FUNCTION_BLOCK FB_String_Test EXTENDS TcUnit.FB_TestSuite

WhenSubtringExistsExpectPosition();
WhenMonthToStringReturnsCorrectMonthName();

METHOD PRIVATE WhenMonthToStringReturnsCorrectMonthName
VAR
    ActualMonth : STRING(10);
    ExpectedMonth : STRING(10) := 'January';
    MTH : INT := 1;
    LANG : INT := 1; // Adjust as needed for your language table
    LX : INT := 0;
END_VAR
TEST(__POUNAME());

// @TEST-RUN
ActualMonth := MONTH_TO_STRING(MTH:=MTH, LANG:=LANG, LX:=LX);

// @TEST-ASSERT
AssertEquals_STRING(ExpectedMonth, ActualMonth, 'MONTH_TO_STRING did not return expected month name');

TEST_FINISHED();
END_METHOD

METHOD PRIVATE WhenSubtringExistsExpectPosition
VAR
	ActualPosition : INT;
	ExpectedPosition : INT := 11;
END_VAR
TEST(__POUNAME());

// @TEST-RUN
ActualPosition := FINDP(str:='Premature optimization is the root of all evil', src:='optimization', pos:=1);

// @TEST-ASSERT
AssertTrue(ActualPosition=ExpectedPosition, 'Substring not found in target string');

TEST_FINISHED();
END_METHOD

END_FUNCTION_BLOCK

(* stored: Version 1.1.0.1
   POU FB_String_Test: Id {7fbd58cc-a844-42ef-9dfc-37fe675b9be6}, SpecialFunc None
   Method WhenMonthToStringReturnsCorrectMonthName: Id {4be9c321-14b4-4109-98ef-f805349c3ea1}
   Method WhenSubtringExistsExpectPosition: Id {f43cd479-0c2b-4ed5-ab04-cc6edd49aa4c} *)
